PROGRAM TELNET_LOG_DEMO
VAR
	TELNET_LOG: TELNET_LOG;
	IPC: IP_C;
	S_BUF: NETWORK_BUFFER;
	R_BUF: NETWORK_BUFFER;
	READY: BOOL;
	IP_CONTROL: IP_CONTROL;
	TON_1: TON;
	LOG_MSG: LOG_MSG;
END_VAR

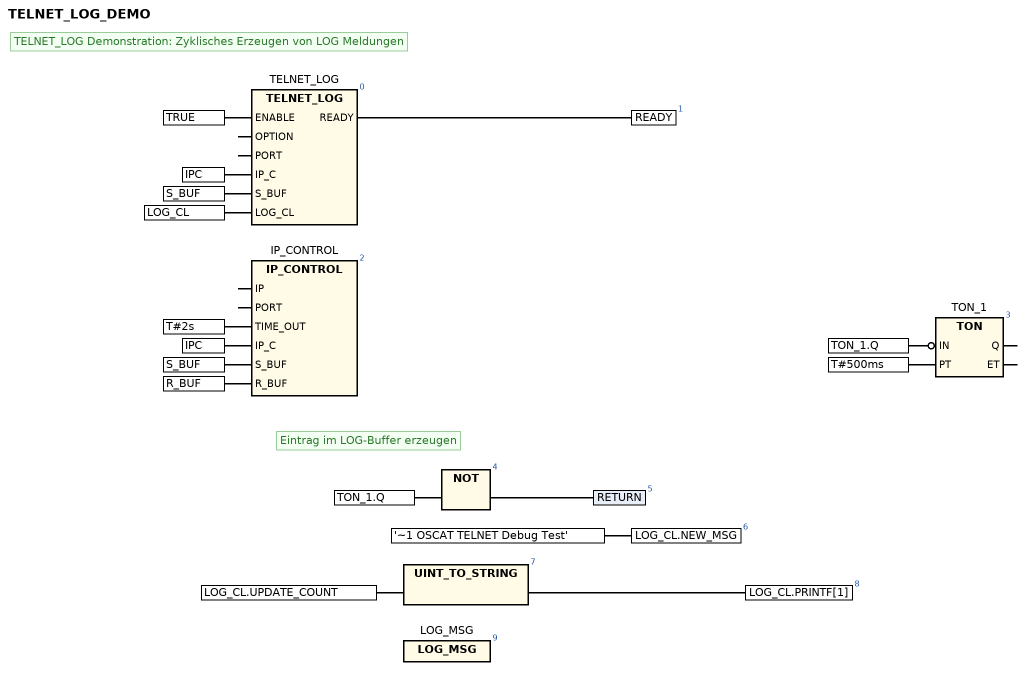
// TELNET_LOG Demonstration: Zyklisches Erzeugen von LOG Meldungen
TELNET_LOG(ENABLE := TRUE, IP_C := IPC, S_BUF := S_BUF, LOG_CL := LOG_CL);
READY := TELNET_LOG.READY;
IP_CONTROL(TIME_OUT := T#2s, IP_C := IPC, S_BUF := S_BUF, R_BUF := R_BUF);
TON_1(IN := NOT TON_1.Q, PT := T#500ms); // TON
// Eintrag im LOG-Buffer erzeugen
IF NOT TON_1.Q THEN RETURN; END_IF
LOG_CL.NEW_MSG := '~1 OSCAT TELNET Debug Test';
LOG_CL.PRINTF[1] := UINT_TO_STRING(LOG_CL.UPDATE_COUNT);
LOG_MSG();

END_PROGRAM

(* stored: Version 1.1.0.1, ProductVersion 3.1.4024.9
   POU TELNET_LOG_DEMO: Id {902389e6-0b1e-4523-906d-01b921020e20}, SpecialFunc None *)
